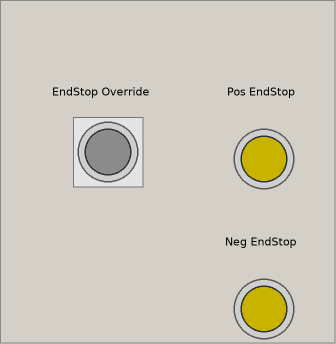
VISUALIZATION HMI  // 336x344
    PushSwitch (73,117 70x70), variable: HMI.bEndStopOverride, behaviour: TOGGLE, style: Switch-PushSwitch-Gray
    Lamp1 (229,124 70x70), variable: P_Outputs.bEndStopPosActive, style: Lamp-Lamp1-Yellow
    Label (26,77 150x30), "EndStop Override"
    Label (186,77 150x30), "Pos EndStop"
    Lamp1 (229,274 70x70), variable: P_Outputs.bEndStopNegActive, style: Lamp-Lamp1-Yellow
    Label (186,227 150x30), "Neg EndStop"
END_VISUALIZATION

(* stored: Version 1.1.0.1, ProductVersion 3.1.4026.11
   Visu HMI: Id {7753864f-df6f-4a20-8851-17b344b9d768} *)
